// CODESYS_Control_for_Raspberry_Pi/Application/visualization/ups_s2/ups_s2_m3_state
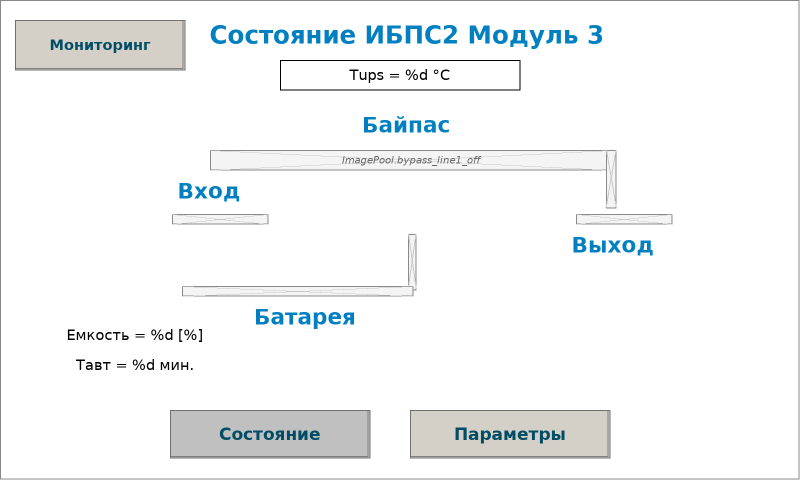
VISUALIZATION ups_s2_m3_state  // 800x480, background image ImagePool.mpx_state_bg
    Rectangle (204,20 406x30), "Состояние ИБПС2 Модуль 3"
    Button (410,410 200x48), "Параметры"
        OnMouseClick:  Assign=ups_s2_m3_params, Type=Assignment
    Button (170,410 200x48), "Состояние", pressed state: PLC_PRG.var_true
    Rectangle (350,110 112x30), "Байпас"
    Rectangle (246,302 118x30), "Батарея"
    Rectangle (166,176 86x30), "Вход"
    Rectangle (560,230 106x30), "Выход"
    Rectangle (280,60 240x30), "Tups = %d °С", text variable: PLC_PRG.mpx_s2_3_temp
    Rectangle (30,320 210x30), "Емкость = %d [%]", text variable: PLC_PRG.mpx_s2_3_battery_capacity
    Rectangle (30,350 210x30), "Tавт = %d мин.", text variable: PLC_PRG.mpx_s2_3_battery_time
    Image (210,150 402x20), image: ImagePool.bypass_line1_off
        p84334746: PLC_PRG.mpx_s2_3_bypass_line_state
    Image (606,150 10x58), image: ImagePool.bypass_arrow_off
        p84334746: PLC_PRG.mpx_s2_3_bypass_arrow_state
    Image (576,214 96x10), image: ImagePool.arrow_off
        p84334746: PLC_PRG.mpx_s2_3_output_state
    Image (172,214 96x10), image: ImagePool.arrow_off
        p84334746: PLC_PRG.mpx_s2_3_input_state
    Image (408,234 8x56), image: ImagePool.battery_arrow_off
        p84334746: PLC_PRG.mpx_s2_3_battery_arrow_state
    Image (182,286 231x10), image: ImagePool.battery_line_off
        p84334746: PLC_PRG.mpx_s2_3_battery_line_state
    Button (15,20 170x50), "Мониторинг"
        OnMouseClick:  Assign=monitoring, Type=Assignment
    hotkey  Id=481037385728, Key=KeyDown=True, KeyName=0, VisuElemId=38
    hotkey  Id=481038434304, Key=KeyName=0, VisuElemId=38
END_VISUALIZATION

// CODESYS_Control_for_Raspberry_Pi/Application/visualization/ups_s1/ups_s1
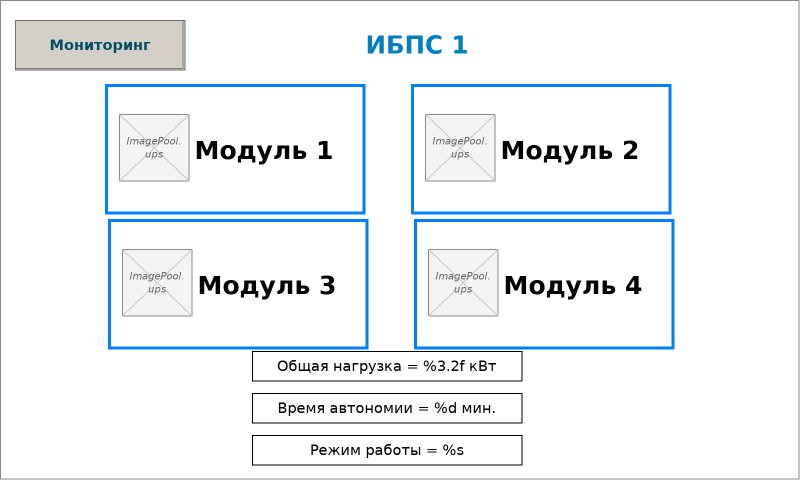
VISUALIZATION ups_s1  // 800x480, background image ImagePool.bg_800
    Group (108,219 260x115)
        OnMouseClick:  Assign=ups_s1_m3_state, Type=Assignment
        RoundedRectangle (0,0 260x130), colour toggle: InterviewState.MPX_S1_3_State
        Image (14,30 70x67), image: ImagePool.ups
        RoundedRectangle (80,38 158x56), "Модуль 3"
            OnMouseClick:  Assign=ups_s2_m1_state, Type=Assignment
    Group (105,84 260x115)
        OnMouseClick:  Assign=ups_s1_m1_state, Type=Assignment
        RoundedRectangle (0,0 260x130), colour toggle: InterviewState.MPX_S1_1_State
        Image (14,30 70x67), image: ImagePool.ups
        RoundedRectangle (80,38 158x56), "Модуль 1"
            OnMouseClick:  Assign=ups_s2_m1_state, Type=Assignment
    Group (414,219 260x115)
        OnMouseClick:  Assign=ups_s1_m4_state, Type=Assignment
        RoundedRectangle (0,0 260x130), colour toggle: InterviewState.MPX_S1_4_State
        Image (14,30 70x67), image: ImagePool.ups
        RoundedRectangle (80,38 158x56), "Модуль 4"
            OnMouseClick:  Assign=ups_s2_m1_state, Type=Assignment
    Group (411,84 260x115)
        OnMouseClick:  Assign=ups_s1_m2_state, Type=Assignment
        RoundedRectangle (0,0 260x130), colour toggle: InterviewState.MPX_S1_2_State
        Image (14,30 70x67), image: ImagePool.ups
        RoundedRectangle (80,38 158x56), "Модуль 2"
            OnMouseClick:  Assign=ups_s2_m1_state, Type=Assignment
    Rectangle (214,30 406x30), "ИБПС 1"
    Button (15,20 170x50), "Мониторинг"
        OnMouseClick:  Assign=monitoring, Type=Assignment
    Rectangle (252,351 270x30), "Общая нагрузка = %3.2f кВт", text variable: PLC_PRG.mpx_s1_all_power
    Rectangle (252,393 270x30), "Время автономии = %d мин.", text variable: PLC_PRG.mpx_s1_1_battery_time
    Rectangle (252,435 270x30), "Режим работы = %s", text variable: PLC_PRG.mpx_s1_state_string
    hotkey  Id=481037385728, Key=KeyDown=True, KeyName=0, VisuElemId=38
    hotkey  Id=481038434304, Key=KeyName=0, VisuElemId=38
END_VISUALIZATION

// CODESYS_Control_for_Raspberry_Pi/Application/visualization/ups_s1/ups_s1_m1_params
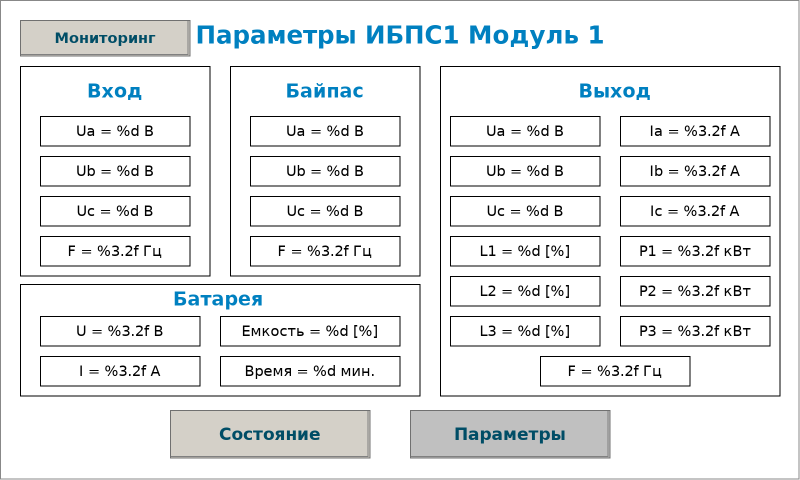
VISUALIZATION ups_s1_m1_params  // 800x480, background image ImagePool.bg_800
    Rectangle (186,20 428x30), "Параметры ИБПC1 Модуль 1"
    Button (170,410 200x48), "Состояние"
        OnMouseClick:  Assign=ups_s1_m1_state, Type=Assignment
    Button (410,410 200x48), "Параметры", pressed state: PLC_PRG.var_true
    Button (20,20 170x36), "Мониторинг"
        OnMouseClick:  Assign=monitoring, Type=Assignment
    Rectangle (20,66 190x210)
    Rectangle (440,66 340x330)
    Rectangle (30,76 170x30), "Вход"
    Rectangle (40,116 150x30), "Ua = %d В", text variable: PLC_PRG.mpx_s1_1_in_v_1
    Rectangle (40,156 150x30), "Ub = %d В", text variable: PLC_PRG.mpx_s1_1_in_v_2
    Rectangle (40,196 150x30), "Uc = %d В", text variable: PLC_PRG.mpx_s1_1_in_v_3
    Rectangle (40,236 150x30), "F = %3.2f Гц", text variable: PLC_PRG.mpx_s1_1_in_freq_real
    Rectangle (230,66 190x210)
    Rectangle (240,76 170x30), "Байпас"
    Rectangle (250,116 150x30), "Ua = %d В", text variable: PLC_PRG.mpx_s1_1_bypass_v_1
    Rectangle (250,156 150x30), "Ub = %d В", text variable: PLC_PRG.mpx_s1_1_bypass_v_2
    Rectangle (250,196 150x30), "Uc = %d В", text variable: PLC_PRG.mpx_s1_1_bypass_v_3
    Rectangle (250,236 150x30), "F = %3.2f Гц", text variable: PLC_PRG.mpx_s1_1_bypass_freq_real
    Rectangle (460,76 310x30), "Выход"
    Rectangle (450,116 150x30), "Ua = %d В", text variable: PLC_PRG.mpx_s1_1_output_v_1
    Rectangle (450,156 150x30), "Ub = %d В", text variable: PLC_PRG.mpx_s1_1_output_v_2
    Rectangle (450,196 150x30), "Uc = %d В", text variable: PLC_PRG.mpx_s1_1_output_v_3
    Rectangle (620,116 150x30), "Ia = %3.2f A", text variable: PLC_PRG.mpx_s1_1_output_i_1_real
    Rectangle (620,156 150x30), "Ib = %3.2f A", text variable: PLC_PRG.mpx_s1_1_output_i_2_real
    Rectangle (620,196 150x30), "Ic = %3.2f A", text variable: PLC_PRG.mpx_s1_1_output_i_3_real
    Rectangle (450,236 150x30), "L1 = %d [%]", text variable: PLC_PRG.mpx_s1_1_load_ph_1
    Rectangle (450,276 150x30), "L2 = %d [%]", text variable: PLC_PRG.mpx_s1_1_load_ph_2
    Rectangle (450,316 150x30), "L3 = %d [%]", text variable: PLC_PRG.mpx_s1_1_load_ph_3
    Rectangle (620,236 150x30), "P1 = %3.2f кВт", text variable: PLC_PRG.mpx_s1_1_output_active_power_1_real
    Rectangle (620,276 150x30), "P2 = %3.2f кВт", text variable: PLC_PRG.mpx_s1_1_output_active_power_2_real
    Rectangle (620,316 150x30), "P3 = %3.2f кВт", text variable: PLC_PRG.mpx_s1_1_output_active_power_3_real
    Rectangle (540,356 150x30), "F = %3.2f Гц", text variable: PLC_PRG.mpx_s1_1_output_freq_real
    Rectangle (20,284 400x112)
    Rectangle (30,290 376x18), "Батарея"
    Rectangle (40,316 160x30), "U = %3.2f В", text variable: PLC_PRG.mpx_s1_1_battery_voltage_real
    Rectangle (40,356 160x30), "I = %3.2f A", text variable: PLC_PRG.mpx_s1_1_battery_current_real
    Rectangle (220,316 180x30), "Емкость = %d [%]", text variable: PLC_PRG.mpx_s1_1_battery_capacity
    Rectangle (220,356 180x30), "Время = %d мин.", text variable: PLC_PRG.mpx_s1_1_battery_time
    hotkey  Id=481037385728, Key=KeyDown=True, KeyName=0, VisuElemId=7
    hotkey  Id=481038434304, Key=KeyName=0, VisuElemId=7
END_VISUALIZATION

// CODESYS_Control_for_Raspberry_Pi/Application/visualization/ups_s1/ups_s1_m1_state
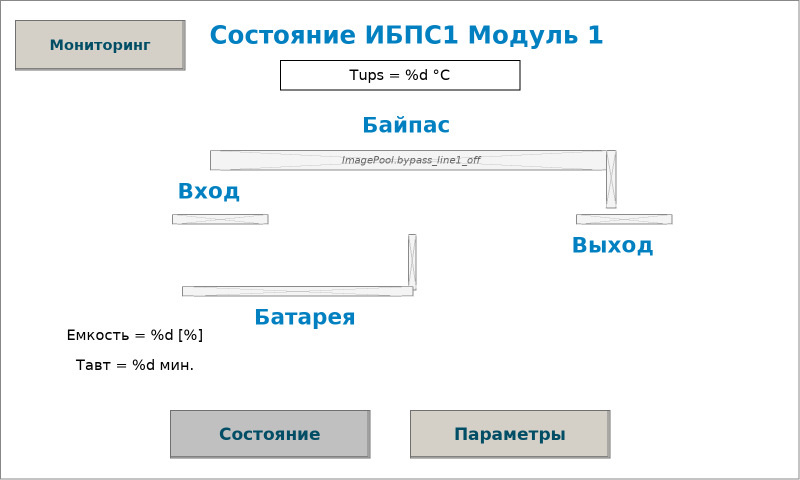
VISUALIZATION ups_s1_m1_state  // 800x480, background image ImagePool.mpx_state_bg
    Rectangle (204,20 406x30), "Состояние ИБПС1 Модуль 1"
    Button (410,410 200x48), "Параметры"
        OnMouseClick:  Assign=ups_s1_m1_params, Type=Assignment
    Button (170,410 200x48), "Состояние", pressed state: PLC_PRG.var_true
    Rectangle (350,110 112x30), "Байпас"
    Rectangle (246,302 118x30), "Батарея"
    Rectangle (166,176 86x30), "Вход"
    Rectangle (560,230 106x30), "Выход"
    Rectangle (280,60 240x30), "Tups = %d °С", text variable: PLC_PRG.mpx_s1_1_temp
    Rectangle (30,320 210x30), "Емкость = %d [%]", text variable: PLC_PRG.mpx_s1_1_battery_capacity
    Rectangle (30,350 210x30), "Tавт = %d мин.", text variable: PLC_PRG.mpx_s1_1_battery_time
    Image (210,150 402x20), image: ImagePool.bypass_line1_off
        p84334746: PLC_PRG.mpx_s1_1_bypass_line_state
    Image (606,150 10x58), image: ImagePool.bypass_arrow_off
        p84334746: PLC_PRG.mpx_s1_1_bypass_arrow_state
    Image (576,214 96x10), image: ImagePool.arrow_off
        p84334746: PLC_PRG.mpx_s1_1_output_state
    Image (172,214 96x10), image: ImagePool.arrow_off
        p84334746: PLC_PRG.mpx_s1_1_input_state
    Image (408,234 8x56), image: ImagePool.battery_arrow_off
        p84334746: PLC_PRG.mpx_s1_1_battery_arrow_state
    Image (182,286 231x10), image: ImagePool.battery_line_off
        p84334746: PLC_PRG.mpx_s1_1_battery_line_state
    Button (15,20 170x50), "Мониторинг"
        OnMouseClick:  Assign=monitoring, Type=Assignment
    hotkey  Id=481037385728, Key=KeyDown=True, KeyName=0, VisuElemId=38
    hotkey  Id=481038434304, Key=KeyName=0, VisuElemId=38
END_VISUALIZATION

// CODESYS_Control_for_Raspberry_Pi/Application/visualization/ups_s1/ups_s1_m2_params
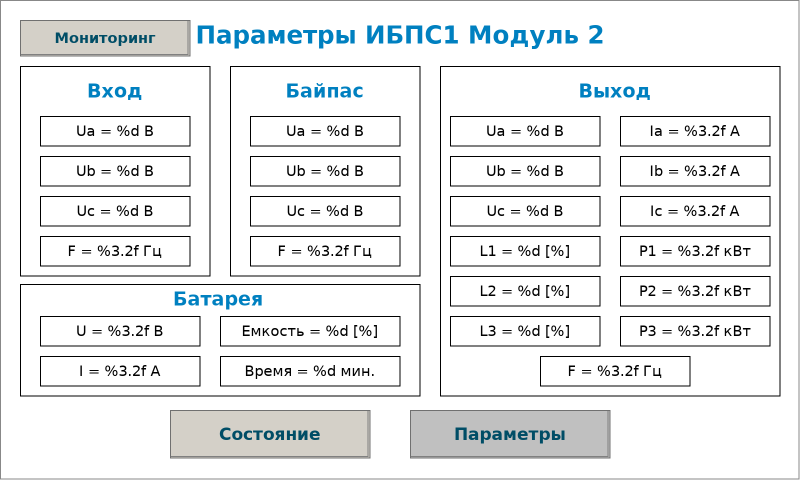
VISUALIZATION ups_s1_m2_params  // 800x480, background image ImagePool.bg_800
    Rectangle (186,20 428x30), "Параметры ИБПC1 Модуль 2"
    Button (170,410 200x48), "Состояние"
        OnMouseClick:  Assign=ups_s1_m2_state, Type=Assignment
    Button (410,410 200x48), "Параметры", pressed state: PLC_PRG.var_true
    Button (20,20 170x36), "Мониторинг"
        OnMouseClick:  Assign=monitoring, Type=Assignment
    Rectangle (20,66 190x210)
    Rectangle (440,66 340x330)
    Rectangle (30,76 170x30), "Вход"
    Rectangle (40,116 150x30), "Ua = %d В", text variable: PLC_PRG.mpx_s1_2_in_v_1
    Rectangle (40,156 150x30), "Ub = %d В", text variable: PLC_PRG.mpx_s1_2_in_v_2
    Rectangle (40,196 150x30), "Uc = %d В", text variable: PLC_PRG.mpx_s1_2_in_v_3
    Rectangle (40,236 150x30), "F = %3.2f Гц", text variable: PLC_PRG.mpx_s1_2_in_freq_real
    Rectangle (230,66 190x210)
    Rectangle (240,76 170x30), "Байпас"
    Rectangle (250,116 150x30), "Ua = %d В", text variable: PLC_PRG.mpx_s1_2_bypass_v_1
    Rectangle (250,156 150x30), "Ub = %d В", text variable: PLC_PRG.mpx_s1_2_bypass_v_2
    Rectangle (250,196 150x30), "Uc = %d В", text variable: PLC_PRG.mpx_s1_2_bypass_v_3
    Rectangle (250,236 150x30), "F = %3.2f Гц", text variable: PLC_PRG.mpx_s1_2_bypass_freq_real
    Rectangle (460,76 310x30), "Выход"
    Rectangle (450,116 150x30), "Ua = %d В", text variable: PLC_PRG.mpx_s1_2_output_v_1
    Rectangle (450,156 150x30), "Ub = %d В", text variable: PLC_PRG.mpx_s1_2_output_v_2
    Rectangle (450,196 150x30), "Uc = %d В", text variable: PLC_PRG.mpx_s1_2_output_v_3
    Rectangle (620,116 150x30), "Ia = %3.2f A", text variable: PLC_PRG.mpx_s1_2_output_i_1_real
    Rectangle (620,156 150x30), "Ib = %3.2f A", text variable: PLC_PRG.mpx_s1_2_output_i_2_real
    Rectangle (620,196 150x30), "Ic = %3.2f A", text variable: PLC_PRG.mpx_s1_2_output_i_3_real
    Rectangle (450,236 150x30), "L1 = %d [%]", text variable: PLC_PRG.mpx_s1_2_load_ph_1
    Rectangle (450,276 150x30), "L2 = %d [%]", text variable: PLC_PRG.mpx_s1_2_load_ph_2
    Rectangle (450,316 150x30), "L3 = %d [%]", text variable: PLC_PRG.mpx_s1_2_load_ph_3
    Rectangle (620,236 150x30), "P1 = %3.2f кВт", text variable: PLC_PRG.mpx_s1_2_output_active_power_1_real
    Rectangle (620,276 150x30), "P2 = %3.2f кВт", text variable: PLC_PRG.mpx_s1_2_output_active_power_2_real
    Rectangle (620,316 150x30), "P3 = %3.2f кВт", text variable: PLC_PRG.mpx_s1_2_output_active_power_3_real
    Rectangle (540,356 150x30), "F = %3.2f Гц", text variable: PLC_PRG.mpx_s1_2_output_freq_real
    Rectangle (20,284 400x112)
    Rectangle (30,290 376x18), "Батарея"
    Rectangle (40,316 160x30), "U = %3.2f В", text variable: PLC_PRG.mpx_s1_2_battery_voltage_real
    Rectangle (40,356 160x30), "I = %3.2f A", text variable: PLC_PRG.mpx_s1_2_battery_current_real
    Rectangle (220,316 180x30), "Емкость = %d [%]", text variable: PLC_PRG.mpx_s1_2_battery_capacity
    Rectangle (220,356 180x30), "Время = %d мин.", text variable: PLC_PRG.mpx_s1_2_battery_time
    hotkey  Id=481037385728, Key=KeyDown=True, KeyName=0, VisuElemId=7
    hotkey  Id=481038434304, Key=KeyName=0, VisuElemId=7
END_VISUALIZATION

// CODESYS_Control_for_Raspberry_Pi/Application/visualization/ups_s1/ups_s1_m2_state
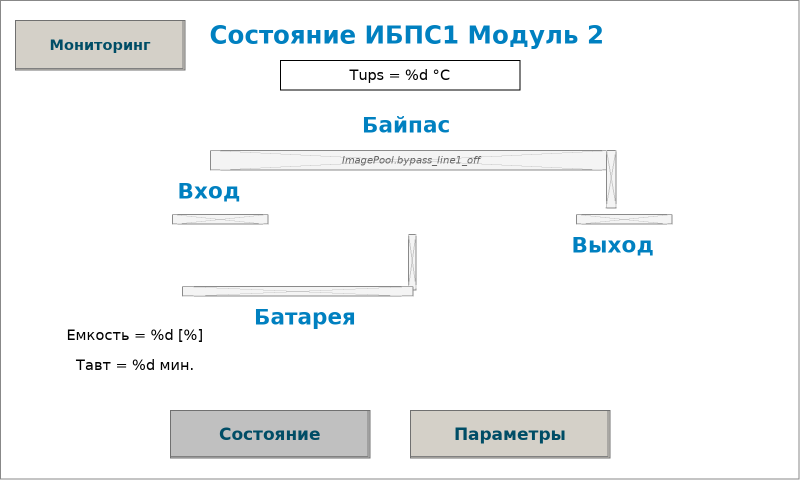
VISUALIZATION ups_s1_m2_state  // 800x480, background image ImagePool.mpx_state_bg
    Rectangle (204,20 406x30), "Состояние ИБПС1 Модуль 2"
    Button (410,410 200x48), "Параметры"
        OnMouseClick:  Assign=ups_s1_m2_params, Type=Assignment
    Button (170,410 200x48), "Состояние", pressed state: PLC_PRG.var_true
    Rectangle (350,110 112x30), "Байпас"
    Rectangle (246,302 118x30), "Батарея"
    Rectangle (166,176 86x30), "Вход"
    Rectangle (560,230 106x30), "Выход"
    Rectangle (280,60 240x30), "Tups = %d °С", text variable: PLC_PRG.mpx_s1_2_temp
    Rectangle (30,320 210x30), "Емкость = %d [%]", text variable: PLC_PRG.mpx_s1_2_battery_capacity
    Rectangle (30,350 210x30), "Tавт = %d мин.", text variable: PLC_PRG.mpx_s1_2_battery_time
    Image (210,150 402x20), image: ImagePool.bypass_line1_off
        p84334746: PLC_PRG.mpx_s1_2_bypass_line_state
    Image (606,150 10x58), image: ImagePool.bypass_arrow_off
        p84334746: PLC_PRG.mpx_s1_2_bypass_arrow_state
    Image (576,214 96x10), image: ImagePool.arrow_off
        p84334746: PLC_PRG.mpx_s1_2_output_state
    Image (172,214 96x10), image: ImagePool.arrow_off
        p84334746: PLC_PRG.mpx_s1_2_input_state
    Image (408,234 8x56), image: ImagePool.battery_arrow_off
        p84334746: PLC_PRG.mpx_s1_2_battery_arrow_state
    Image (182,286 231x10), image: ImagePool.battery_line_off
        p84334746: PLC_PRG.mpx_s1_2_battery_line_state
    Button (15,20 170x50), "Мониторинг"
        OnMouseClick:  Assign=monitoring, Type=Assignment
    hotkey  Id=481037385728, Key=KeyDown=True, KeyName=0, VisuElemId=38
    hotkey  Id=481038434304, Key=KeyName=0, VisuElemId=38
END_VISUALIZATION

// CODESYS_Control_for_Raspberry_Pi/Application/visualization/ups_s1/ups_s1_m3_params
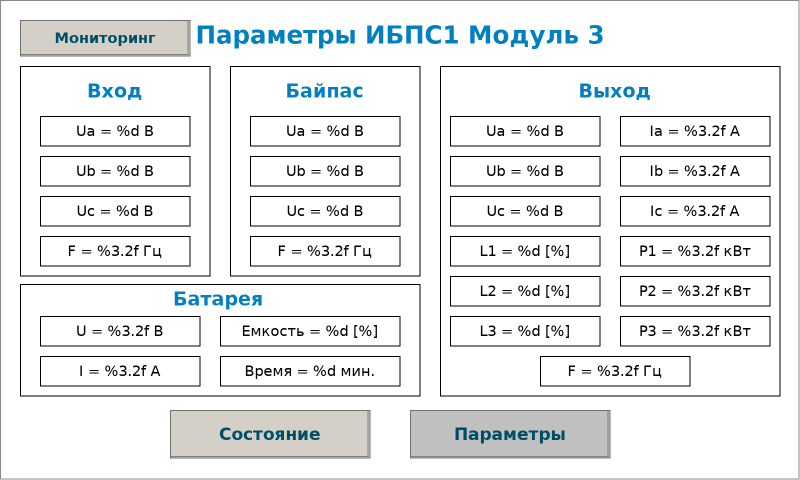
VISUALIZATION ups_s1_m3_params  // 800x480, background image ImagePool.bg_800
    Rectangle (186,20 428x30), "Параметры ИБПC1 Модуль 3"
    Button (170,410 200x48), "Состояние"
        OnMouseClick:  Assign=ups_s1_m3_state, Type=Assignment
    Button (410,410 200x48), "Параметры", pressed state: PLC_PRG.var_true
    Button (20,20 170x36), "Мониторинг"
        OnMouseClick:  Assign=monitoring, Type=Assignment
    Rectangle (20,66 190x210)
    Rectangle (440,66 340x330)
    Rectangle (30,76 170x30), "Вход"
    Rectangle (40,116 150x30), "Ua = %d В", text variable: PLC_PRG.mpx_s1_3_in_v_1
    Rectangle (40,156 150x30), "Ub = %d В", text variable: PLC_PRG.mpx_s1_3_in_v_2
    Rectangle (40,196 150x30), "Uc = %d В", text variable: PLC_PRG.mpx_s1_3_in_v_3
    Rectangle (40,236 150x30), "F = %3.2f Гц", text variable: PLC_PRG.mpx_s1_3_in_freq_real
    Rectangle (230,66 190x210)
    Rectangle (240,76 170x30), "Байпас"
    Rectangle (250,116 150x30), "Ua = %d В", text variable: PLC_PRG.mpx_s1_3_bypass_v_1
    Rectangle (250,156 150x30), "Ub = %d В", text variable: PLC_PRG.mpx_s1_3_bypass_v_2
    Rectangle (250,196 150x30), "Uc = %d В", text variable: PLC_PRG.mpx_s1_3_bypass_v_3
    Rectangle (250,236 150x30), "F = %3.2f Гц", text variable: PLC_PRG.mpx_s1_3_bypass_freq_real
    Rectangle (460,76 310x30), "Выход"
    Rectangle (450,116 150x30), "Ua = %d В", text variable: PLC_PRG.mpx_s1_3_output_v_1
    Rectangle (450,156 150x30), "Ub = %d В", text variable: PLC_PRG.mpx_s1_3_output_v_2
    Rectangle (450,196 150x30), "Uc = %d В", text variable: PLC_PRG.mpx_s1_3_output_v_3
    Rectangle (620,116 150x30), "Ia = %3.2f A", text variable: PLC_PRG.mpx_s1_3_output_i_1_real
    Rectangle (620,156 150x30), "Ib = %3.2f A", text variable: PLC_PRG.mpx_s1_3_output_i_2_real
    Rectangle (620,196 150x30), "Ic = %3.2f A", text variable: PLC_PRG.mpx_s1_3_output_i_3_real
    Rectangle (450,236 150x30), "L1 = %d [%]", text variable: PLC_PRG.mpx_s1_3_load_ph_1
    Rectangle (450,276 150x30), "L2 = %d [%]", text variable: PLC_PRG.mpx_s1_3_load_ph_2
    Rectangle (450,316 150x30), "L3 = %d [%]", text variable: PLC_PRG.mpx_s1_3_load_ph_3
    Rectangle (620,236 150x30), "P1 = %3.2f кВт", text variable: PLC_PRG.mpx_s1_3_output_active_power_1_real
    Rectangle (620,276 150x30), "P2 = %3.2f кВт", text variable: PLC_PRG.mpx_s1_3_output_active_power_2_real
    Rectangle (620,316 150x30), "P3 = %3.2f кВт", text variable: PLC_PRG.mpx_s1_3_output_active_power_3_real
    Rectangle (540,356 150x30), "F = %3.2f Гц", text variable: PLC_PRG.mpx_s1_3_output_freq_real
    Rectangle (20,284 400x112)
    Rectangle (30,290 376x18), "Батарея"
    Rectangle (40,316 160x30), "U = %3.2f В", text variable: PLC_PRG.mpx_s1_3_battery_voltage_real
    Rectangle (40,356 160x30), "I = %3.2f A", text variable: PLC_PRG.mpx_s1_3_battery_current_real
    Rectangle (220,316 180x30), "Емкость = %d [%]", text variable: PLC_PRG.mpx_s1_3_battery_capacity
    Rectangle (220,356 180x30), "Время = %d мин.", text variable: PLC_PRG.mpx_s1_3_battery_time
    hotkey  Id=481037385728, Key=KeyDown=True, KeyName=0, VisuElemId=7
    hotkey  Id=481038434304, Key=KeyName=0, VisuElemId=7
END_VISUALIZATION

// CODESYS_Control_for_Raspberry_Pi/Application/visualization/ups_s1/ups_s1_m3_state
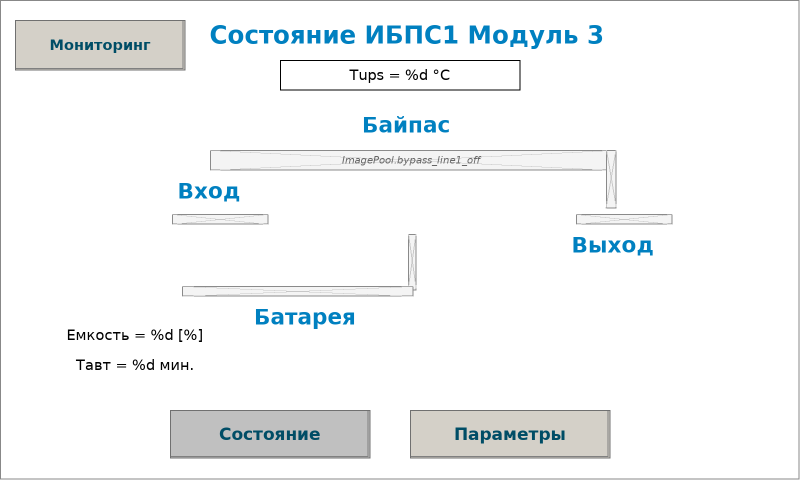
VISUALIZATION ups_s1_m3_state  // 800x480, background image ImagePool.mpx_state_bg
    Rectangle (204,20 406x30), "Состояние ИБПС1 Модуль 3"
    Button (410,410 200x48), "Параметры"
        OnMouseClick:  Assign=ups_s1_m3_params, Type=Assignment
    Button (170,410 200x48), "Состояние", pressed state: PLC_PRG.var_true
    Rectangle (350,110 112x30), "Байпас"
    Rectangle (246,302 118x30), "Батарея"
    Rectangle (166,176 86x30), "Вход"
    Rectangle (560,230 106x30), "Выход"
    Rectangle (280,60 240x30), "Tups = %d °С", text variable: PLC_PRG.mpx_s1_3_temp
    Rectangle (30,320 210x30), "Емкость = %d [%]", text variable: PLC_PRG.mpx_s1_3_battery_capacity
    Rectangle (30,350 210x30), "Tавт = %d мин.", text variable: PLC_PRG.mpx_s1_3_battery_time
    Image (210,150 402x20), image: ImagePool.bypass_line1_off
        p84334746: PLC_PRG.mpx_s1_3_bypass_line_state
    Image (606,150 10x58), image: ImagePool.bypass_arrow_off
        p84334746: PLC_PRG.mpx_s1_3_bypass_arrow_state
    Image (576,214 96x10), image: ImagePool.arrow_off
        p84334746: PLC_PRG.mpx_s1_3_output_state
    Image (172,214 96x10), image: ImagePool.arrow_off
        p84334746: PLC_PRG.mpx_s1_3_input_state
    Image (408,234 8x56), image: ImagePool.battery_arrow_off
        p84334746: PLC_PRG.mpx_s1_3_battery_arrow_state
    Image (182,286 231x10), image: ImagePool.battery_line_off
        p84334746: PLC_PRG.mpx_s1_3_battery_line_state
    Button (15,20 170x50), "Мониторинг"
        OnMouseClick:  Assign=monitoring, Type=Assignment
    hotkey  Id=481037385728, Key=KeyDown=True, KeyName=0, VisuElemId=38
    hotkey  Id=481038434304, Key=KeyName=0, VisuElemId=38
END_VISUALIZATION

// CODESYS_Control_for_Raspberry_Pi/Application/visualization/ups_s1/ups_s1_m4_params
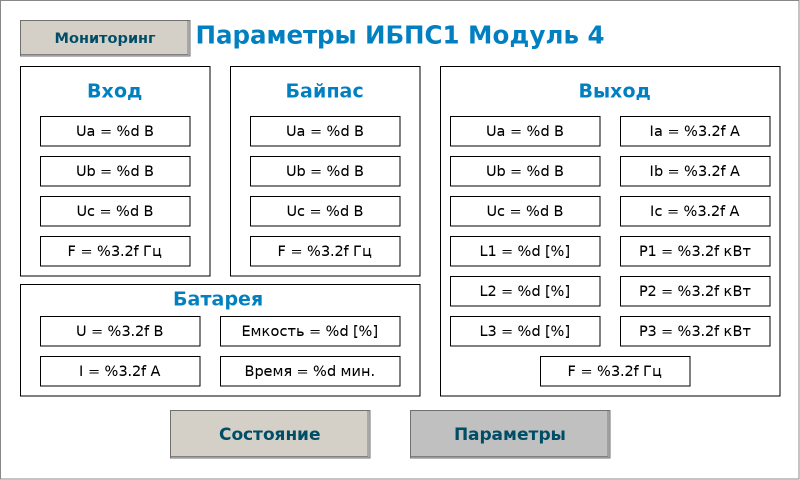
VISUALIZATION ups_s1_m4_params  // 800x480, background image ImagePool.bg_800
    Rectangle (186,20 428x30), "Параметры ИБПC1 Модуль 4"
    Button (170,410 200x48), "Состояние"
        OnMouseClick:  Assign=ups_s1_m4_state, Type=Assignment
    Button (410,410 200x48), "Параметры", pressed state: PLC_PRG.var_true
    Button (20,20 170x36), "Мониторинг"
        OnMouseClick:  Assign=monitoring, Type=Assignment
    Rectangle (20,66 190x210)
    Rectangle (440,66 340x330)
    Rectangle (30,76 170x30), "Вход"
    Rectangle (40,116 150x30), "Ua = %d В", text variable: PLC_PRG.mpx_s1_4_in_v_1
    Rectangle (40,156 150x30), "Ub = %d В", text variable: PLC_PRG.mpx_s1_4_in_v_2
    Rectangle (40,196 150x30), "Uc = %d В", text variable: PLC_PRG.mpx_s1_4_in_v_3
    Rectangle (40,236 150x30), "F = %3.2f Гц", text variable: PLC_PRG.mpx_s1_4_in_freq_real
    Rectangle (230,66 190x210)
    Rectangle (240,76 170x30), "Байпас"
    Rectangle (250,116 150x30), "Ua = %d В", text variable: PLC_PRG.mpx_s1_4_bypass_v_1
    Rectangle (250,156 150x30), "Ub = %d В", text variable: PLC_PRG.mpx_s1_4_bypass_v_2
    Rectangle (250,196 150x30), "Uc = %d В", text variable: PLC_PRG.mpx_s1_4_bypass_v_3
    Rectangle (250,236 150x30), "F = %3.2f Гц", text variable: PLC_PRG.mpx_s1_4_bypass_freq_real
    Rectangle (460,76 310x30), "Выход"
    Rectangle (450,116 150x30), "Ua = %d В", text variable: PLC_PRG.mpx_s1_4_output_v_1
    Rectangle (450,156 150x30), "Ub = %d В", text variable: PLC_PRG.mpx_s1_4_output_v_2
    Rectangle (450,196 150x30), "Uc = %d В", text variable: PLC_PRG.mpx_s1_4_output_v_3
    Rectangle (620,116 150x30), "Ia = %3.2f A", text variable: PLC_PRG.mpx_s1_4_output_i_1_real
    Rectangle (620,156 150x30), "Ib = %3.2f A", text variable: PLC_PRG.mpx_s1_4_output_i_2_real
    Rectangle (620,196 150x30), "Ic = %3.2f A", text variable: PLC_PRG.mpx_s1_4_output_i_3_real
    Rectangle (450,236 150x30), "L1 = %d [%]", text variable: PLC_PRG.mpx_s1_4_load_ph_1
    Rectangle (450,276 150x30), "L2 = %d [%]", text variable: PLC_PRG.mpx_s1_4_load_ph_2
    Rectangle (450,316 150x30), "L3 = %d [%]", text variable: PLC_PRG.mpx_s1_4_load_ph_3
    Rectangle (620,236 150x30), "P1 = %3.2f кВт", text variable: PLC_PRG.mpx_s1_4_output_active_power_1_real
    Rectangle (620,276 150x30), "P2 = %3.2f кВт", text variable: PLC_PRG.mpx_s1_4_output_active_power_2_real
    Rectangle (620,316 150x30), "P3 = %3.2f кВт", text variable: PLC_PRG.mpx_s1_4_output_active_power_3_real
    Rectangle (540,356 150x30), "F = %3.2f Гц", text variable: PLC_PRG.mpx_s1_4_output_freq_real
    Rectangle (20,284 400x112)
    Rectangle (30,290 376x18), "Батарея"
    Rectangle (40,316 160x30), "U = %3.2f В", text variable: PLC_PRG.mpx_s1_4_battery_voltage_real
    Rectangle (40,356 160x30), "I = %3.2f A", text variable: PLC_PRG.mpx_s1_4_battery_current_real
    Rectangle (220,316 180x30), "Емкость = %d [%]", text variable: PLC_PRG.mpx_s1_4_battery_capacity
    Rectangle (220,356 180x30), "Время = %d мин.", text variable: PLC_PRG.mpx_s1_4_battery_time
    hotkey  Id=481037385728, Key=KeyDown=True, KeyName=0, VisuElemId=7
    hotkey  Id=481038434304, Key=KeyName=0, VisuElemId=7
END_VISUALIZATION

// CODESYS_Control_for_Raspberry_Pi/Application/visualization/ups_s1/ups_s1_m4_state
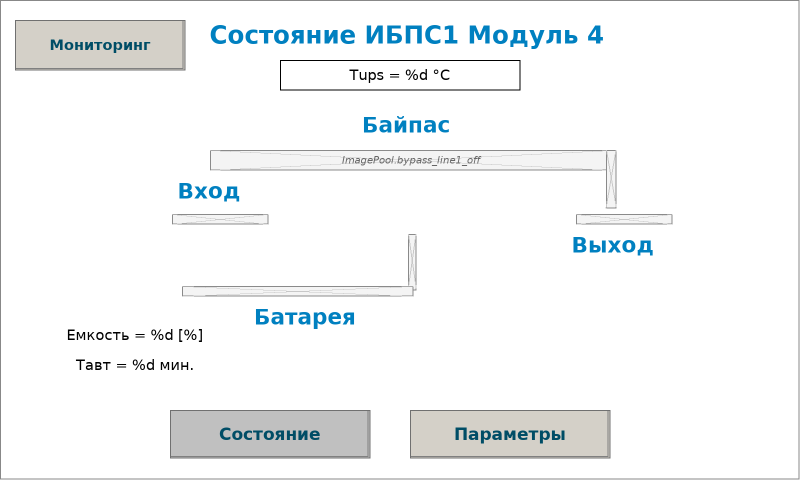
VISUALIZATION ups_s1_m4_state  // 800x480, background image ImagePool.mpx_state_bg
    Rectangle (204,20 406x30), "Состояние ИБПС1 Модуль 4"
    Button (410,410 200x48), "Параметры"
        OnMouseClick:  Assign=ups_s1_m4_params, Type=Assignment
    Button (170,410 200x48), "Состояние", pressed state: PLC_PRG.var_true
    Rectangle (350,110 112x30), "Байпас"
    Rectangle (246,302 118x30), "Батарея"
    Rectangle (166,176 86x30), "Вход"
    Rectangle (560,230 106x30), "Выход"
    Rectangle (280,60 240x30), "Tups = %d °С", text variable: PLC_PRG.mpx_s1_4_temp
    Rectangle (30,320 210x30), "Емкость = %d [%]", text variable: PLC_PRG.mpx_s1_4_battery_capacity
    Rectangle (30,350 210x30), "Tавт = %d мин.", text variable: PLC_PRG.mpx_s1_4_battery_time
    Image (210,150 402x20), image: ImagePool.bypass_line1_off
        p84334746: PLC_PRG.mpx_s1_4_bypass_line_state
    Image (606,150 10x58), image: ImagePool.bypass_arrow_off
        p84334746: PLC_PRG.mpx_s1_4_bypass_arrow_state
    Image (576,214 96x10), image: ImagePool.arrow_off
        p84334746: PLC_PRG.mpx_s1_4_output_state
    Image (172,214 96x10), image: ImagePool.arrow_off
        p84334746: PLC_PRG.mpx_s1_4_input_state
    Image (408,234 8x56), image: ImagePool.battery_arrow_off
        p84334746: PLC_PRG.mpx_s1_4_battery_arrow_state
    Image (182,286 231x10), image: ImagePool.battery_line_off
        p84334746: PLC_PRG.mpx_s1_4_battery_line_state
    Button (15,20 170x50), "Мониторинг"
        OnMouseClick:  Assign=monitoring, Type=Assignment
    hotkey  Id=481037385728, Key=KeyDown=True, KeyName=0, VisuElemId=38
    hotkey  Id=481038434304, Key=KeyName=0, VisuElemId=38
END_VISUALIZATION

// CODESYS_Control_for_Raspberry_Pi/Application/visualization/ups_a1/ups_a1
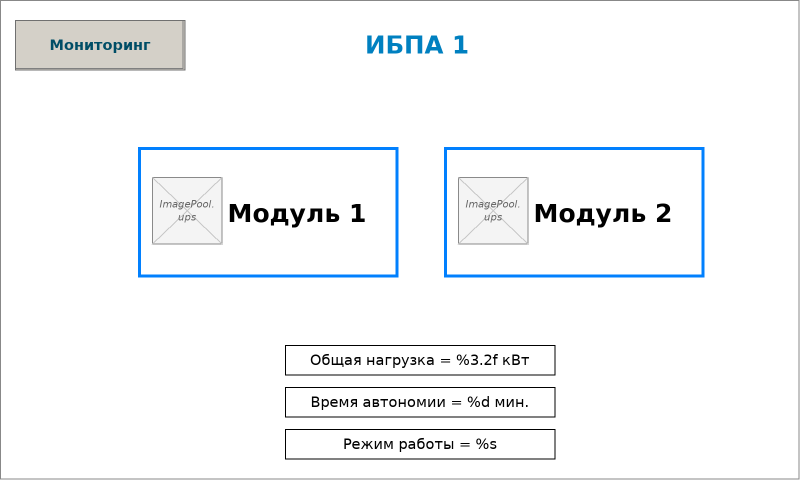
VISUALIZATION ups_a1  // 800x480, background image ImagePool.bg_800
    Rectangle (214,30 406x30), "ИБПА 1"
    Button (15,20 170x50), "Мониторинг"
        OnMouseClick:  Assign=monitoring, Type=Assignment
    Group (138,147 260x115)
        OnMouseClick:  Assign=ups_a1_m1_state, Type=Assignment
        RoundedRectangle (0,0 260x130), colour toggle: InterviewState.MPX_S1_1_State
        Image (14,30 70x67), image: ImagePool.ups
        RoundedRectangle (80,38 158x56), "Модуль 1"
            OnMouseClick:  Assign=ups_s2_m1_state, Type=Assignment
    Group (444,147 260x115)
        OnMouseClick:  Assign=ups_a1_m2_state, Type=Assignment
        RoundedRectangle (0,0 260x130), colour toggle: InterviewState.MPX_S1_2_State
        Image (14,30 70x67), image: ImagePool.ups
        RoundedRectangle (80,38 158x56), "Модуль 2"
            OnMouseClick:  Assign=ups_s2_m1_state, Type=Assignment
    Rectangle (285,345 270x30), "Общая нагрузка = %3.2f кВт", text variable: PLC_PRG.mpx_a1_all_power
    Rectangle (285,387 270x30), "Время автономии = %d мин.", text variable: PLC_PRG.mpx_a1_1_battery_time
    Rectangle (285,429 270x30), "Режим работы = %s", text variable: PLC_PRG.mpx_a1_state_string
    hotkey  Id=481037385728, Key=KeyDown=True, KeyName=0, VisuElemId=38
    hotkey  Id=481038434304, Key=KeyName=0, VisuElemId=38
END_VISUALIZATION

// CODESYS_Control_for_Raspberry_Pi/Application/visualization/ups_a1/ups_a1_m1_params
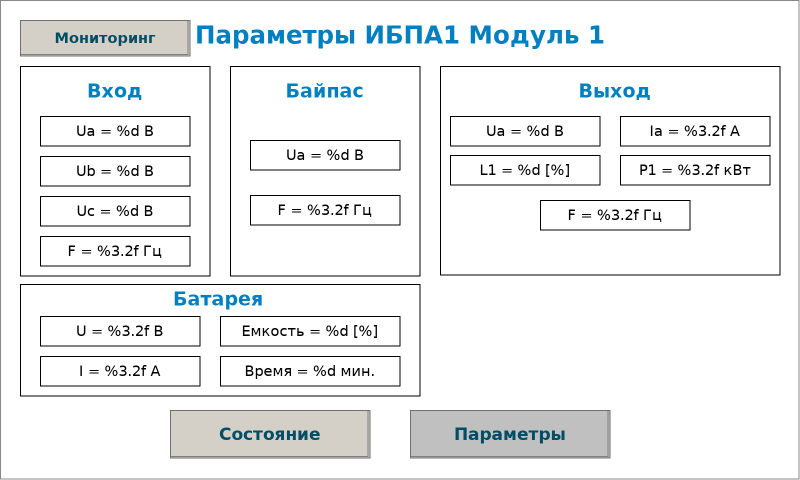
VISUALIZATION ups_a1_m1_params  // 800x480, background image ImagePool.bg_800
    Rectangle (186,20 428x30), "Параметры ИБПА1 Модуль 1"
    Button (170,410 200x48), "Состояние"
        OnMouseClick:  Assign=ups_a1_m1_state, Type=Assignment
    Button (410,410 200x48), "Параметры", pressed state: PLC_PRG.var_true
    Button (20,20 170x36), "Мониторинг"
        OnMouseClick:  Assign=monitoring, Type=Assignment
    Rectangle (20,66 190x210)
    Rectangle (440,66 340x209)
    Rectangle (30,76 170x30), "Вход"
    Rectangle (40,116 150x30), "Ua = %d В", text variable: PLC_PRG.mpx_a1_1_in_v_1
    Rectangle (40,156 150x30), "Ub = %d В", text variable: PLC_PRG.mpx_a1_1_in_v_2
    Rectangle (40,196 150x30), "Uc = %d В", text variable: PLC_PRG.mpx_a1_1_in_v_3
    Rectangle (40,236 150x30), "F = %3.2f Гц", text variable: PLC_PRG.mpx_a1_1_in_freq_real
    Rectangle (230,66 190x210)
    Rectangle (240,76 170x30), "Байпас"
    Rectangle (250,140 150x30), "Ua = %d В", text variable: PLC_PRG.mpx_a1_1_bypass_v_1
    Rectangle (250,195 150x30), "F = %3.2f Гц", text variable: PLC_PRG.mpx_a1_1_bypass_freq_real
    Rectangle (460,76 310x30), "Выход"
    Rectangle (450,116 150x30), "Ua = %d В", text variable: PLC_PRG.mpx_a1_1_output_v_1
    Rectangle (620,116 150x30), "Ia = %3.2f A", text variable: PLC_PRG.mpx_a1_1_output_i_1_real
    Rectangle (450,155 150x30), "L1 = %d [%]", text variable: PLC_PRG.mpx_a1_1_load_ph_1
    Rectangle (620,155 150x30), "P1 = %3.2f кВт", text variable: PLC_PRG.mpx_a1_1_output_active_power_1_real
    Rectangle (540,200 150x30), "F = %3.2f Гц", text variable: PLC_PRG.mpx_a1_1_output_freq_real
    Rectangle (20,284 400x112)
    Rectangle (30,290 376x18), "Батарея"
    Rectangle (40,316 160x30), "U = %3.2f В", text variable: PLC_PRG.mpx_a1_1_battery_voltage_real
    Rectangle (40,356 160x30), "I = %3.2f A", text variable: PLC_PRG.mpx_a1_1_battery_current_real
    Rectangle (220,316 180x30), "Емкость = %d [%]", text variable: PLC_PRG.mpx_a1_1_battery_capacity
    Rectangle (220,356 180x30), "Время = %d мин.", text variable: PLC_PRG.mpx_a1_1_battery_time
    hotkey  Id=481037385728, Key=KeyDown=True, KeyName=0, VisuElemId=7
    hotkey  Id=481038434304, Key=KeyName=0, VisuElemId=7
END_VISUALIZATION

// CODESYS_Control_for_Raspberry_Pi/Application/visualization/ups_a1/ups_a1_m1_state
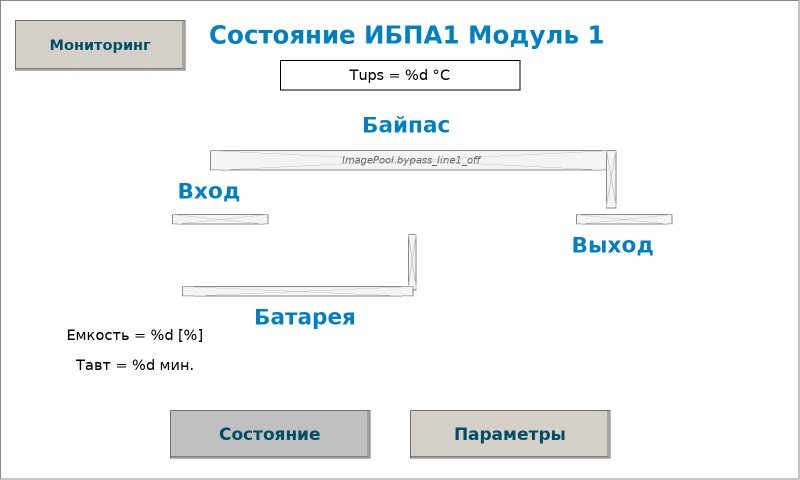
VISUALIZATION ups_a1_m1_state  // 800x480, background image ImagePool.mpx_state_bg
    Rectangle (204,20 406x30), "Состояние ИБПА1 Модуль 1"
    Button (410,410 200x48), "Параметры"
        OnMouseClick:  Assign=ups_a1_m1_params, Type=Assignment
    Button (170,410 200x48), "Состояние", pressed state: PLC_PRG.var_true
    Rectangle (350,110 112x30), "Байпас"
    Rectangle (246,302 118x30), "Батарея"
    Rectangle (166,176 86x30), "Вход"
    Rectangle (560,230 106x30), "Выход"
    Rectangle (280,60 240x30), "Tups = %d °С", text variable: PLC_PRG.mpx_a1_1_temp
    Rectangle (30,320 210x30), "Емкость = %d [%]", text variable: PLC_PRG.mpx_a1_1_battery_capacity
    Rectangle (30,350 210x30), "Tавт = %d мин.", text variable: PLC_PRG.mpx_a1_1_battery_time
    Image (210,150 402x20), image: ImagePool.bypass_line1_off
        p84334746: PLC_PRG.mpx_a1_1_bypass_line_state
    Image (606,150 10x58), image: ImagePool.bypass_arrow_off
        p84334746: PLC_PRG.mpx_a1_1_bypass_arrow_state
    Image (576,214 96x10), image: ImagePool.arrow_off
        p84334746: PLC_PRG.mpx_a1_1_output_state
    Image (172,214 96x10), image: ImagePool.arrow_off
        p84334746: PLC_PRG.mpx_a1_1_input_state
    Image (408,234 8x56), image: ImagePool.battery_arrow_off
        p84334746: PLC_PRG.mpx_a1_1_battery_arrow_state
    Image (182,286 231x10), image: ImagePool.battery_line_off
        p84334746: PLC_PRG.mpx_a1_1_battery_line_state
    Button (15,20 170x50), "Мониторинг"
        OnMouseClick:  Assign=monitoring, Type=Assignment
    hotkey  Id=481037385728, Key=KeyDown=True, KeyName=0, VisuElemId=38
    hotkey  Id=481038434304, Key=KeyName=0, VisuElemId=38
END_VISUALIZATION

// CODESYS_Control_for_Raspberry_Pi/Application/visualization/ups_a1/ups_a1_m2_params
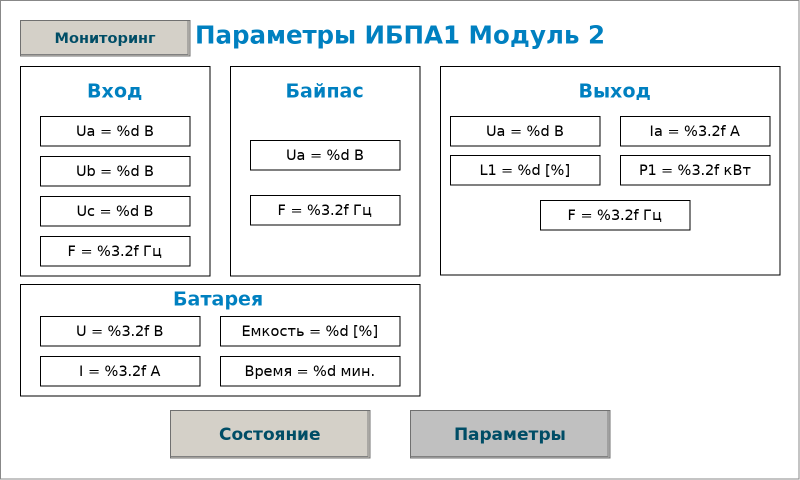
VISUALIZATION ups_a1_m2_params  // 800x480, background image ImagePool.bg_800
    Rectangle (186,20 428x30), "Параметры ИБПА1 Модуль 2"
    Button (170,410 200x48), "Состояние"
        OnMouseClick:  Assign=ups_a1_m2_state, Type=Assignment
    Button (410,410 200x48), "Параметры", pressed state: PLC_PRG.var_true
    Button (20,20 170x36), "Мониторинг"
        OnMouseClick:  Assign=monitoring, Type=Assignment
    Rectangle (20,66 190x210)
    Rectangle (440,66 340x209)
    Rectangle (30,76 170x30), "Вход"
    Rectangle (40,116 150x30), "Ua = %d В", text variable: PLC_PRG.mpx_a1_2_in_v_1
    Rectangle (40,156 150x30), "Ub = %d В", text variable: PLC_PRG.mpx_a1_2_in_v_2
    Rectangle (40,196 150x30), "Uc = %d В", text variable: PLC_PRG.mpx_a1_2_in_v_3
    Rectangle (40,236 150x30), "F = %3.2f Гц", text variable: PLC_PRG.mpx_a1_2_in_freq_real
    Rectangle (230,66 190x210)
    Rectangle (240,76 170x30), "Байпас"
    Rectangle (250,140 150x30), "Ua = %d В", text variable: PLC_PRG.mpx_a1_2_bypass_v_1
    Rectangle (250,195 150x30), "F = %3.2f Гц", text variable: PLC_PRG.mpx_a1_2_bypass_freq_real
    Rectangle (460,76 310x30), "Выход"
    Rectangle (450,116 150x30), "Ua = %d В", text variable: PLC_PRG.mpx_a1_2_output_v_1
    Rectangle (620,116 150x30), "Ia = %3.2f A", text variable: PLC_PRG.mpx_a1_2_output_i_1_real
    Rectangle (450,155 150x30), "L1 = %d [%]", text variable: PLC_PRG.mpx_a1_2_load_ph_1
    Rectangle (620,155 150x30), "P1 = %3.2f кВт", text variable: PLC_PRG.mpx_a1_2_output_active_power_1_real
    Rectangle (540,200 150x30), "F = %3.2f Гц", text variable: PLC_PRG.mpx_a1_2_output_freq_real
    Rectangle (20,284 400x112)
    Rectangle (30,290 376x18), "Батарея"
    Rectangle (40,316 160x30), "U = %3.2f В", text variable: PLC_PRG.mpx_a1_2_battery_voltage_real
    Rectangle (40,356 160x30), "I = %3.2f A", text variable: PLC_PRG.mpx_a1_2_battery_current_real
    Rectangle (220,316 180x30), "Емкость = %d [%]", text variable: PLC_PRG.mpx_a1_2_battery_capacity
    Rectangle (220,356 180x30), "Время = %d мин.", text variable: PLC_PRG.mpx_a1_2_battery_time
    hotkey  Id=481037385728, Key=KeyDown=True, KeyName=0, VisuElemId=7
    hotkey  Id=481038434304, Key=KeyName=0, VisuElemId=7
END_VISUALIZATION

// CODESYS_Control_for_Raspberry_Pi/Application/visualization/ups_a1/ups_a1_m2_state
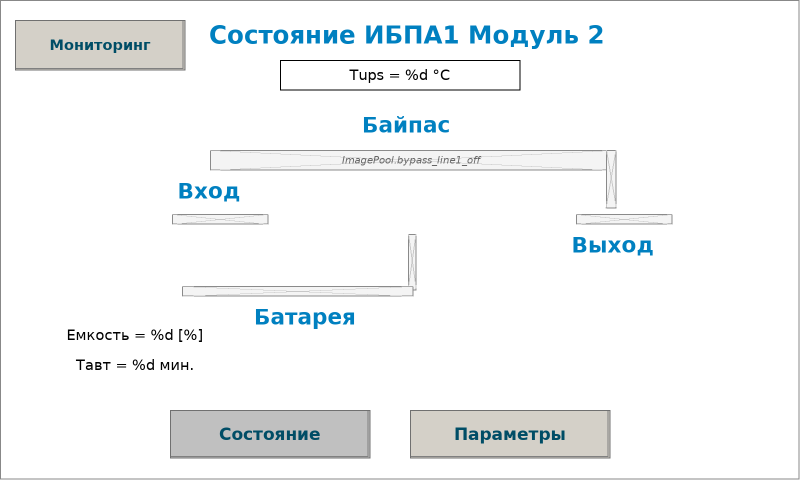
VISUALIZATION ups_a1_m2_state  // 800x480, background image ImagePool.mpx_state_bg
    Rectangle (204,20 406x30), "Состояние ИБПА1 Модуль 2"
    Button (410,410 200x48), "Параметры"
        OnMouseClick:  Assign=ups_a1_m2_params, Type=Assignment
    Button (170,410 200x48), "Состояние", pressed state: PLC_PRG.var_true
    Rectangle (350,110 112x30), "Байпас"
    Rectangle (246,302 118x30), "Батарея"
    Rectangle (166,176 86x30), "Вход"
    Rectangle (560,230 106x30), "Выход"
    Rectangle (280,60 240x30), "Tups = %d °С", text variable: PLC_PRG.mpx_a1_2_temp
    Rectangle (30,320 210x30), "Емкость = %d [%]", text variable: PLC_PRG.mpx_a1_2_battery_capacity
    Rectangle (30,350 210x30), "Tавт = %d мин.", text variable: PLC_PRG.mpx_a1_2_battery_time
    Image (210,150 402x20), image: ImagePool.bypass_line1_off
        p84334746: PLC_PRG.mpx_a1_2_bypass_line_state
    Image (606,150 10x58), image: ImagePool.bypass_arrow_off
        p84334746: PLC_PRG.mpx_a1_2_bypass_arrow_state
    Image (576,214 96x10), image: ImagePool.arrow_off
        p84334746: PLC_PRG.mpx_a1_2_output_state
    Image (172,214 96x10), image: ImagePool.arrow_off
        p84334746: PLC_PRG.mpx_a1_2_input_state
    Image (408,234 8x56), image: ImagePool.battery_arrow_off
        p84334746: PLC_PRG.mpx_a1_2_battery_arrow_state
    Image (182,286 231x10), image: ImagePool.battery_line_off
        p84334746: PLC_PRG.mpx_a1_2_battery_line_state
    Button (15,20 170x50), "Мониторинг"
        OnMouseClick:  Assign=monitoring, Type=Assignment
    hotkey  Id=481037385728, Key=KeyDown=True, KeyName=0, VisuElemId=38
    hotkey  Id=481038434304, Key=KeyName=0, VisuElemId=38
END_VISUALIZATION

// CODESYS_Control_for_Raspberry_Pi/Application/visualization/ups_a2/ups_a2
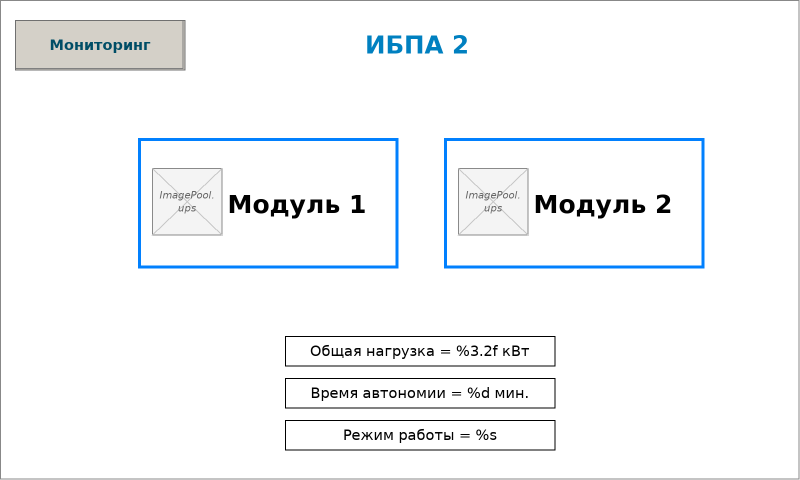
VISUALIZATION ups_a2  // 800x480, background image ImagePool.bg_800
    Rectangle (214,30 406x30), "ИБПА 2"
    Button (15,20 170x50), "Мониторинг"
        OnMouseClick:  Assign=monitoring, Type=Assignment
    Group (138,138 260x115)
        OnMouseClick:  Assign=ups_a2_m1_state, Type=Assignment
        RoundedRectangle (0,0 260x130), colour toggle: InterviewState.MPX_S1_1_State
        Image (14,30 70x67), image: ImagePool.ups
        RoundedRectangle (80,38 158x56), "Модуль 1"
            OnMouseClick:  Assign=ups_s2_m1_state, Type=Assignment
    Group (444,138 260x115)
        OnMouseClick:  Assign=ups_a2_m2_state, Type=Assignment
        RoundedRectangle (0,0 260x130), colour toggle: InterviewState.MPX_S1_2_State
        Image (14,30 70x67), image: ImagePool.ups
        RoundedRectangle (80,38 158x56), "Модуль 2"
            OnMouseClick:  Assign=ups_s2_m1_state, Type=Assignment
    Rectangle (285,336 270x30), "Общая нагрузка = %3.2f кВт", text variable: PLC_PRG.mpx_a2_all_power
    Rectangle (285,378 270x30), "Время автономии = %d мин.", text variable: PLC_PRG.mpx_a2_1_battery_time
    Rectangle (285,420 270x30), "Режим работы = %s", text variable: PLC_PRG.mpx_a2_state_string
    hotkey  Id=481037385728, Key=KeyDown=True, KeyName=0, VisuElemId=38
    hotkey  Id=481038434304, Key=KeyName=0, VisuElemId=38
END_VISUALIZATION

// CODESYS_Control_for_Raspberry_Pi/Application/visualization/ups_a2/ups_a2_m1_params
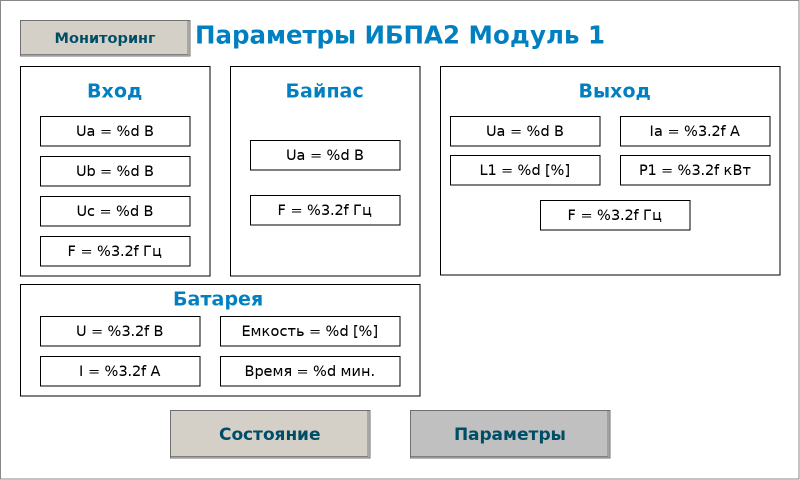
VISUALIZATION ups_a2_m1_params  // 800x480, background image ImagePool.bg_800
    Rectangle (186,20 428x30), "Параметры ИБПА2 Модуль 1"
    Button (170,410 200x48), "Состояние"
        OnMouseClick:  Assign=ups_a2_m1_state, Type=Assignment
    Button (410,410 200x48), "Параметры", pressed state: PLC_PRG.var_true
    Button (20,20 170x36), "Мониторинг"
        OnMouseClick:  Assign=monitoring, Type=Assignment
    Rectangle (20,66 190x210)
    Rectangle (440,66 340x209)
    Rectangle (30,76 170x30), "Вход"
    Rectangle (40,116 150x30), "Ua = %d В", text variable: PLC_PRG.mpx_a2_1_in_v_1
    Rectangle (40,156 150x30), "Ub = %d В", text variable: PLC_PRG.mpx_a2_1_in_v_2
    Rectangle (40,196 150x30), "Uc = %d В", text variable: PLC_PRG.mpx_a2_1_in_v_3
    Rectangle (40,236 150x30), "F = %3.2f Гц", text variable: PLC_PRG.mpx_a2_1_in_freq_real
    Rectangle (230,66 190x210)
    Rectangle (240,76 170x30), "Байпас"
    Rectangle (250,140 150x30), "Ua = %d В", text variable: PLC_PRG.mpx_a2_1_bypass_v_1
    Rectangle (250,195 150x30), "F = %3.2f Гц", text variable: PLC_PRG.mpx_a2_1_bypass_freq_real
    Rectangle (460,76 310x30), "Выход"
    Rectangle (450,116 150x30), "Ua = %d В", text variable: PLC_PRG.mpx_a2_1_output_v_1
    Rectangle (620,116 150x30), "Ia = %3.2f A", text variable: PLC_PRG.mpx_a2_1_output_i_1_real
    Rectangle (450,155 150x30), "L1 = %d [%]", text variable: PLC_PRG.mpx_a2_1_load_ph_1
    Rectangle (620,155 150x30), "P1 = %3.2f кВт", text variable: PLC_PRG.mpx_a2_1_output_active_power_1_real
    Rectangle (540,200 150x30), "F = %3.2f Гц", text variable: PLC_PRG.mpx_a2_1_output_freq_real
    Rectangle (20,284 400x112)
    Rectangle (30,290 376x18), "Батарея"
    Rectangle (40,316 160x30), "U = %3.2f В", text variable: PLC_PRG.mpx_a2_1_battery_voltage_real
    Rectangle (40,356 160x30), "I = %3.2f A", text variable: PLC_PRG.mpx_a2_1_battery_current_real
    Rectangle (220,316 180x30), "Емкость = %d [%]", text variable: PLC_PRG.mpx_a2_1_battery_capacity
    Rectangle (220,356 180x30), "Время = %d мин.", text variable: PLC_PRG.mpx_a2_1_battery_time
    hotkey  Id=481037385728, Key=KeyDown=True, KeyName=0, VisuElemId=7
    hotkey  Id=481038434304, Key=KeyName=0, VisuElemId=7
END_VISUALIZATION

// CODESYS_Control_for_Raspberry_Pi/Application/visualization/ups_a2/ups_a2_m1_state
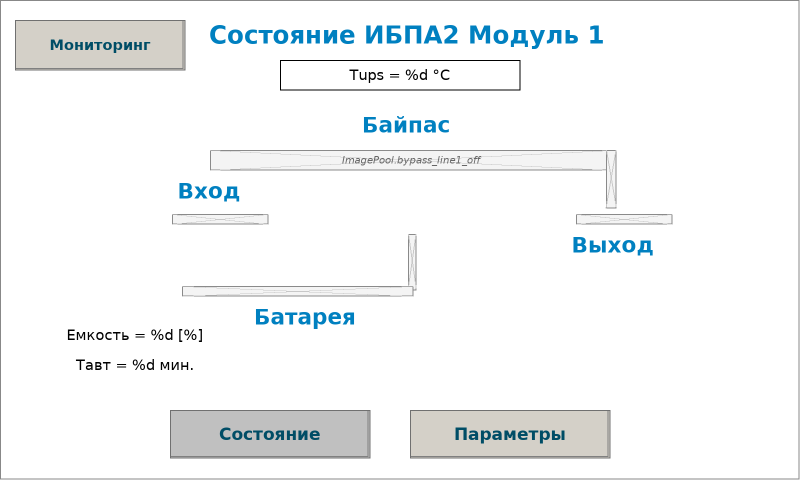
VISUALIZATION ups_a2_m1_state  // 800x480, background image ImagePool.mpx_state_bg
    Rectangle (204,20 406x30), "Состояние ИБПА2 Модуль 1"
    Button (410,410 200x48), "Параметры"
        OnMouseClick:  Assign=ups_a2_m1_params, Type=Assignment
    Button (170,410 200x48), "Состояние", pressed state: PLC_PRG.var_true
    Rectangle (350,110 112x30), "Байпас"
    Rectangle (246,302 118x30), "Батарея"
    Rectangle (166,176 86x30), "Вход"
    Rectangle (560,230 106x30), "Выход"
    Rectangle (280,60 240x30), "Tups = %d °С", text variable: PLC_PRG.mpx_a2_1_temp
    Rectangle (30,320 210x30), "Емкость = %d [%]", text variable: PLC_PRG.mpx_a2_1_battery_capacity
    Rectangle (30,350 210x30), "Tавт = %d мин.", text variable: PLC_PRG.mpx_a2_1_battery_time
    Image (210,150 402x20), image: ImagePool.bypass_line1_off
        p84334746: PLC_PRG.mpx_a2_1_bypass_line_state
    Image (606,150 10x58), image: ImagePool.bypass_arrow_off
        p84334746: PLC_PRG.mpx_a2_1_bypass_arrow_state
    Image (576,214 96x10), image: ImagePool.arrow_off
        p84334746: PLC_PRG.mpx_a2_1_output_state
    Image (172,214 96x10), image: ImagePool.arrow_off
        p84334746: PLC_PRG.mpx_a2_1_input_state
    Image (408,234 8x56), image: ImagePool.battery_arrow_off
        p84334746: PLC_PRG.mpx_a2_1_battery_arrow_state
    Image (182,286 231x10), image: ImagePool.battery_line_off
        p84334746: PLC_PRG.mpx_a2_1_battery_line_state
    Button (15,20 170x50), "Мониторинг"
        OnMouseClick:  Assign=monitoring, Type=Assignment
    hotkey  Id=481037385728, Key=KeyDown=True, KeyName=0, VisuElemId=38
    hotkey  Id=481038434304, Key=KeyName=0, VisuElemId=38
END_VISUALIZATION

// CODESYS_Control_for_Raspberry_Pi/Application/visualization/ups_a2/ups_a2_m2_params
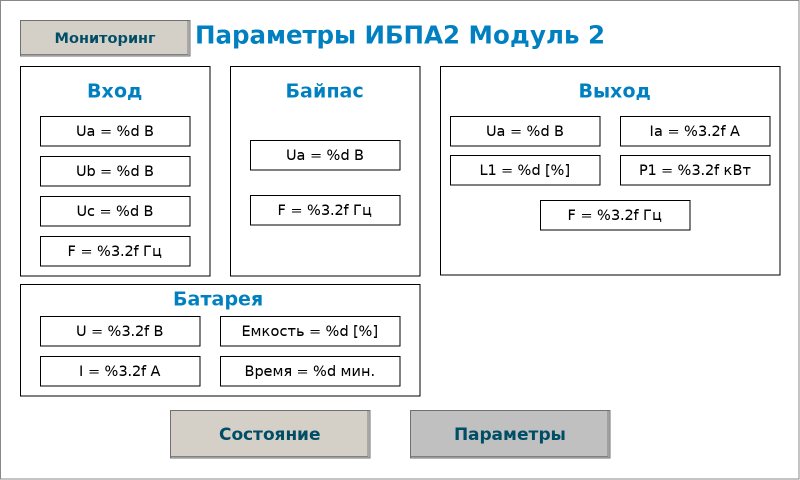
VISUALIZATION ups_a2_m2_params  // 800x480, background image ImagePool.bg_800
    Rectangle (186,20 428x30), "Параметры ИБПА2 Модуль 2"
    Button (170,410 200x48), "Состояние"
        OnMouseClick:  Assign=ups_a2_m2_state, Type=Assignment
    Button (410,410 200x48), "Параметры", pressed state: PLC_PRG.var_true
    Button (20,20 170x36), "Мониторинг"
        OnMouseClick:  Assign=monitoring, Type=Assignment
    Rectangle (20,66 190x210)
    Rectangle (440,66 340x209)
    Rectangle (30,76 170x30), "Вход"
    Rectangle (40,116 150x30), "Ua = %d В", text variable: PLC_PRG.mpx_a2_2_in_v_1
    Rectangle (40,156 150x30), "Ub = %d В", text variable: PLC_PRG.mpx_a2_2_in_v_2
    Rectangle (40,196 150x30), "Uc = %d В", text variable: PLC_PRG.mpx_a2_2_in_v_3
    Rectangle (40,236 150x30), "F = %3.2f Гц", text variable: PLC_PRG.mpx_a2_2_in_freq_real
    Rectangle (230,66 190x210)
    Rectangle (240,76 170x30), "Байпас"
    Rectangle (250,140 150x30), "Ua = %d В", text variable: PLC_PRG.mpx_a2_2_bypass_v_1
    Rectangle (250,195 150x30), "F = %3.2f Гц", text variable: PLC_PRG.mpx_a2_2_bypass_freq_real
    Rectangle (460,76 310x30), "Выход"
    Rectangle (450,116 150x30), "Ua = %d В", text variable: PLC_PRG.mpx_a2_2_output_v_1
    Rectangle (620,116 150x30), "Ia = %3.2f A", text variable: PLC_PRG.mpx_a2_2_output_i_1_real
    Rectangle (450,155 150x30), "L1 = %d [%]", text variable: PLC_PRG.mpx_a2_2_load_ph_1
    Rectangle (620,155 150x30), "P1 = %3.2f кВт", text variable: PLC_PRG.mpx_a2_2_output_active_power_1_real
    Rectangle (540,200 150x30), "F = %3.2f Гц", text variable: PLC_PRG.mpx_a2_2_output_freq_real
    Rectangle (20,284 400x112)
    Rectangle (30,290 376x18), "Батарея"
    Rectangle (40,316 160x30), "U = %3.2f В", text variable: PLC_PRG.mpx_a2_2_battery_voltage_real
    Rectangle (40,356 160x30), "I = %3.2f A", text variable: PLC_PRG.mpx_a2_2_battery_current_real
    Rectangle (220,316 180x30), "Емкость = %d [%]", text variable: PLC_PRG.mpx_a2_2_battery_capacity
    Rectangle (220,356 180x30), "Время = %d мин.", text variable: PLC_PRG.mpx_a2_2_battery_time
    hotkey  Id=481037385728, Key=KeyDown=True, KeyName=0, VisuElemId=7
    hotkey  Id=481038434304, Key=KeyName=0, VisuElemId=7
END_VISUALIZATION

// CODESYS_Control_for_Raspberry_Pi/Application/visualization/ups_a2/ups_a2_m2_state
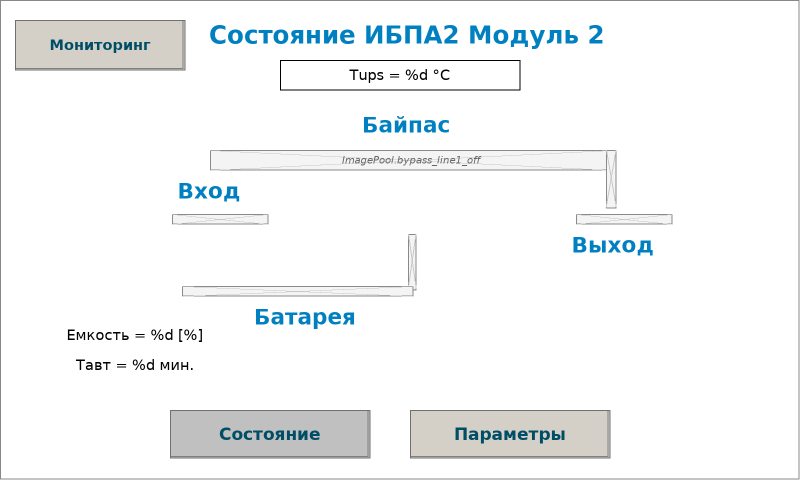
VISUALIZATION ups_a2_m2_state  // 800x480, background image ImagePool.mpx_state_bg
    Rectangle (204,20 406x30), "Состояние ИБПА2 Модуль 2"
    Button (410,410 200x48), "Параметры"
        OnMouseClick:  Assign=ups_a2_m2_params, Type=Assignment
    Button (170,410 200x48), "Состояние", pressed state: PLC_PRG.var_true
    Rectangle (350,110 112x30), "Байпас"
    Rectangle (246,302 118x30), "Батарея"
    Rectangle (166,176 86x30), "Вход"
    Rectangle (560,230 106x30), "Выход"
    Rectangle (280,60 240x30), "Tups = %d °С", text variable: PLC_PRG.mpx_a2_2_temp
    Rectangle (30,320 210x30), "Емкость = %d [%]", text variable: PLC_PRG.mpx_a2_2_battery_capacity
    Rectangle (30,350 210x30), "Tавт = %d мин.", text variable: PLC_PRG.mpx_a2_2_battery_time
    Image (210,150 402x20), image: ImagePool.bypass_line1_off
        p84334746: PLC_PRG.mpx_a2_2_bypass_line_state
    Image (606,150 10x58), image: ImagePool.bypass_arrow_off
        p84334746: PLC_PRG.mpx_a2_2_bypass_arrow_state
    Image (576,214 96x10), image: ImagePool.arrow_off
        p84334746: PLC_PRG.mpx_a2_2_output_state
    Image (172,214 96x10), image: ImagePool.arrow_off
        p84334746: PLC_PRG.mpx_a2_2_input_state
    Image (408,234 8x56), image: ImagePool.battery_arrow_off
        p84334746: PLC_PRG.mpx_a2_2_battery_arrow_state
    Image (182,286 231x10), image: ImagePool.battery_line_off
        p84334746: PLC_PRG.mpx_a2_2_battery_line_state
    Button (15,20 170x50), "Мониторинг"
        OnMouseClick:  Assign=monitoring, Type=Assignment
    hotkey  Id=481037385728, Key=KeyDown=True, KeyName=0, VisuElemId=38
    hotkey  Id=481038434304, Key=KeyName=0, VisuElemId=38
END_VISUALIZATION

// CODESYS_Control_for_Raspberry_Pi/Application/visualization/climate_log
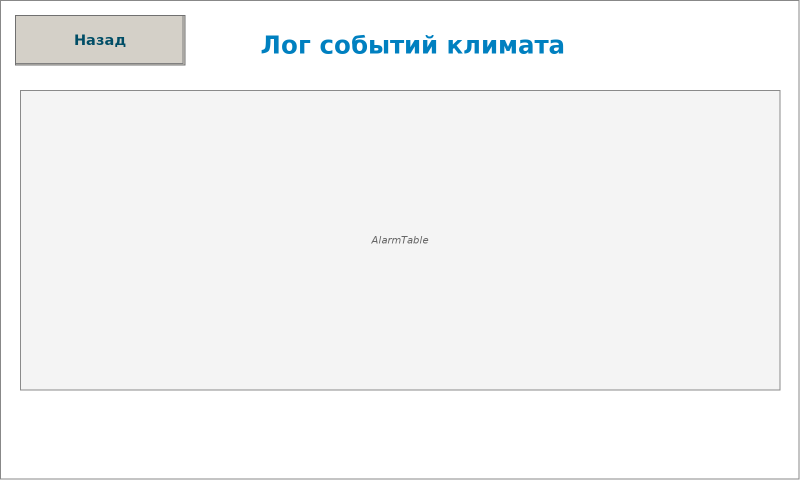
VISUALIZATION climate_log  // 800x480, background image ImagePool.bg_800
    Button (15,15 170x50), "Назад"
        OnMouseClick:  Assign=climate, Type=Previous
    Rectangle (210,30 406x30), "Лог событий климата"
    AlarmTable (20,90 760x300)
        Column[0]: ColumnTitle=Временная отметка
        Column[1]: ColumnTitle=Сообщение
        p1521930926: ClimateGroup
        p1663851261: __All
        p3266827225: PLC_PRG.var_true
    hotkey  Id=481037385728, Key=KeyDown=True, KeyName=0, VisuElemId=1
    hotkey  Id=481038434304, Key=KeyName=0, VisuElemId=1
END_VISUALIZATION

// CODESYS_Control_for_Raspberry_Pi/Application/visualization/more
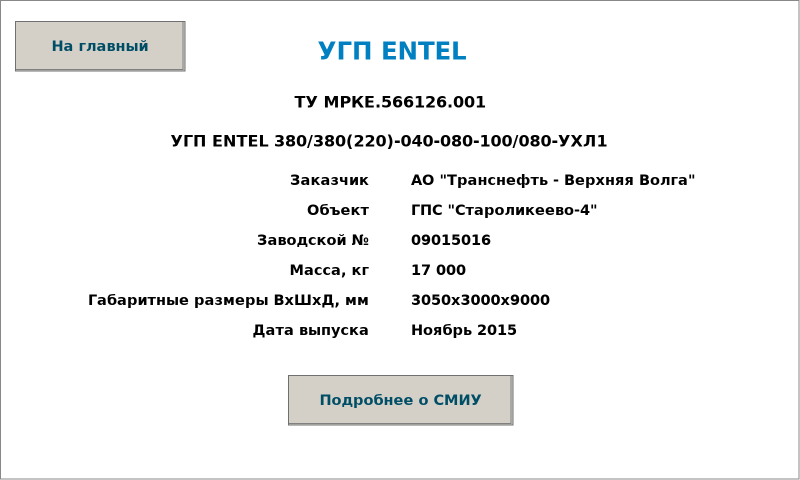
VISUALIZATION more  // 800x480, background image ImagePool.bg_800
    Rectangle (189,36 406x30), "УГП ENTEL"
    Button (15,21 170x50), "На главный"
        OnMouseClick:  Assign=main, Type=Assignment
    Button (288,375 225x50), "Подробнее о СМИУ"
        OnMouseClick:  Assign=info, Type=Assignment
    Label (213,87 355x30), "ТУ МРКЕ.566126.001"
    Label (186,126 406x30), "УГП ENTEL 380/380(220)-040-080-100/080-УХЛ1"
    Label (276,165 96x30), "Заказчик"
    Label (276,195 96x30), "Объект"
    Label (246,225 126x30), "Заводской №"
    Label (276,255 96x30), "Масса, кг"
    Label (96,285 276x30), "Габаритные размеры ВхШхД, мм"
    Label (201,315 171x30), "Дата выпуска"
    Label (408,165 309x30), "АО "Транснефть - Верхняя Волга""
    Label (408,195 228x30), "ГПС "Староликеево-4""
    Label (408,225 114x30), "09015016"
    Label (408,255 120x30), "17 000"
    Label (408,285 165x30), "3050х3000х9000"
    Label (408,315 126x30), "Ноябрь 2015"
    hotkey  Id=481037385728, Key=KeyDown=True, KeyName=0, VisuElemId=3
    hotkey  Id=481038434304, Key=KeyName=0, VisuElemId=3
    hotkey  Id=481037385728, Key=KeyDown=True, KeyName=0, VisuElemId=5
    hotkey  Id=481038434304, Key=KeyName=0, VisuElemId=5
END_VISUALIZATION

(* text list AlarmGroup (id | default)
  95 | Отсутствует напряжение на выходе ИБПА 2
  94 | Отсутствует напряжение на выходе ИБПА 1
  93 | Отсутствует напряжение на выходе ИБПС 2
  92 | Отсутствует напряжение на выходе ИБПС 1
  91 | Отсутствует напряжение на входе ИБПА 2
  90 | Отсутствует напряжение на входе ИБПА 1
  89 | Отсутствует напряжение на входе ИБПС 2
  88 | Отсутствует напряжение на входе ИБПС 1
  87 | Отключен выходной автомат ИБПС 2
  86 | Отсутствует напряжения на выходе ИБПС 2 модуль 4 (1ф.)
  85 | Отключен выходной автомат ИБПС 1
  84 | Отсутствует напряжения на выходе ИБПС 2 модуль 4 (3ф.)
  83 | Отсутствует напряжения на выходе ИБПС 2 модуль 4 (2ф.)
  82 | Отсутствует напряжения на выходе ИБПС 2 модуль 4 (1ф.)
  81 | Отсутствует напряжения на выходе ИБПС 2 модуль 3 (3ф.)
  80 | Отсутствует напряжения на выходе ИБПС 2 модуль 3 (2ф.)
  79 | Отсутствует напряжения на выходе ИБПС 2 модуль 3 (1ф.)
  78 | Отсутствует напряжения на выходе ИБПС 2 модуль 2 (3ф.)
  77 | Отсутствует напряжения на выходе ИБПС 2 модуль 2 (2ф.)
  76 | Отсутствует напряжения на выходе ИБПС 2 модуль 2 (1ф.)
  75 | Отсутствует напряжения на выходе ИБПС 2 модуль 1 (3ф.)
  74 | Отсутствует напряжения на выходе ИБПС 2 модуль 1 (2ф.)
  73 | Отсутствует напряжения на выходе ИБПС 2 модуль 1 (1ф.)
  72 | Отсутствует напряжения на выходе ИБПС 1 модуль 4 (3ф.)
  71 | Отсутствует напряжения на выходе ИБПС 1 модуль 4 (2ф.)
  70 | Отсутствует напряжения на выходе ИБПС 1 модуль 4 (1ф.)
  69 | Отсутствует напряжения на выходе ИБПС 1 модуль 3 (3ф.)
  68 | Отсутствует напряжения на выходе ИБПС 1 модуль 3 (2ф.)
  67 | Отсутствует напряжения на выходе ИБПС 1 модуль 3 (1ф.)
  66 | Отсутствует напряжения на выходе ИБПС 1 модуль 2 (3ф.)
  65 | Отсутствует напряжения на выходе ИБПС 1 модуль 2 (2ф.)
  64 | Отсутствует напряжения на выходе ИБПС 1 модуль 2 (1ф.)
  63 | Отсутствует напряжения на выходе ИБПС 1 модуль 1 (3ф.)
  62 | Отсутствует напряжения на выходе ИБПС 1 модуль 1 (2ф.)
  61 | Отсутствует напряжения на выходе ИБПС 1 модуль 1 (1ф.)
  60 | Отсутствует напряжения на выходе ИБПА 2 модуль 2
  59 | Отсутствует напряжения на выходе ИБПА 2 модуль 1
  58 | Отсутствует напряжения на выходе ИБПА 1 модуль 2
  57 | Отсутствует напряжения на выходе ИБПА 1 модуль 1
  56 | Авария ИБПС 2 модуль 4
  55 | Авария ИБПС 2 модуль 3
  54 | Авария ИБПС 2 модуль 2
  53 | Авария ИБПС 2 модуль 1
  52 | Авария ИБПС 1 модуль 4
  51 | Авария ИБПС 1 модуль 3
  50 | Авария ИБПС 1 модуль 2
  49 | Авария ИБПС 1 модуль 1
  48 | Авария ИБПА 2 модуль 2
  47 | Авария ИБПА 2 модуль 1
  46 | Авария ИБПА 1 модуль 2
  45 | Авария ИБПА 1 модуль 1
  44 | Отсутствует напряжение на входе ИБПC 2 модуль 4 (3 ф.)
  43 | Отсутствует напряжение на входе ИБПC 2 модуль 4 (2 ф.)
  42 | Отсутствует напряжение на входе ИБПC 2 модуль 4 (1 ф.)
  41 | Отсутствует напряжение на входе ИБПC 2 модуль 3 (3 ф.)
  40 | Отсутствует напряжение на входе ИБПC 2 модуль 3 (2 ф.)
  39 | Отсутствует напряжение на входе ИБПC 2 модуль 3 (1 ф.)
  38 | Отсутствует напряжение на входе ИБПC 2 модуль 2 (3 ф.)
  37 | Отсутствует напряжение на входе ИБПC 2 модуль 2 (2 ф.)
  36 | Отсутствует напряжение на входе ИБПC 2 модуль 2 (1 ф.)
  35 | Отсутствует напряжение на входе ИБПC 2 модуль 1 (3 ф.)
  34 | Отсутствует напряжение на входе ИБПC 2 модуль 1 (2 ф.)
  33 | Отсутствует напряжение на входе ИБПC 2 модуль 1 (1 ф.)
  32 | Отсутствует напряжение на входе ИБПC 1 модуль 4 (3 ф.)
  31 | Отсутствует напряжение на входе ИБПC 1 модуль 4 (2 ф.)
  30 | Отсутствует напряжение на входе ИБПC 1 модуль 4 (1 ф.)
  29 | Отсутствует напряжение на входе ИБПC 1 модуль 3 (3 ф.)
  28 | Отсутствует напряжение на входе ИБПC 1 модуль 3 (2 ф.)
  27 | Отсутствует напряжение на входе ИБПC 1 модуль 3 (1 ф.)
  26 | Отсутствует напряжение на входе ИБПC 1 модуль 2 (3 ф.)
  25 | Отсутствует напряжение на входе ИБПC 1 модуль 2 (2 ф.)
  24 | Отсутствует напряжение на входе ИБПC 1 модуль 1 (3 ф.)
  23 | Отсутствует напряжение на входе ИБПC 1 модуль 2 (1 ф.)
  22 | Отсутствует напряжение на входе ИБПC 1 модуль 1 (2 ф.)
  21 | Отсутствует напряжение на входе ИБПC 1 модуль 1 (1 ф.)
  20 | Отсутствует напряжение на входе ИБПА 2 модуль 2 (3 ф.)
  19 | Отсутствует напряжение на входе ИБПА 2 модуль 2 (2 ф.)
  18 | Отсутствует напряжение на входе ИБПА 2 модуль 2 (1 ф.)
  17 | Отсутствует напряжение на входе ИБПА 2 модуль 1 (3 ф.)
  16 | Отсутствует напряжение на входе ИБПА 2 модуль 1 (2 ф.)
  15 | Отсутствует напряжение на входе ИБПА 2 модуль 1 (1 ф.)
  14 | Отсутствует напряжение на входе ИБПА 1 модуль 2 (3 ф.)
  13 | Отсутствует напряжение на входе ИБПА 1 модуль 2 (2 ф.)
  12 | Отсутствует напряжение на входе ИБПА 1 модуль 2 (1 ф.)
  11 | Отсутствует напряжение на входе ИБПА 1 модуль 1 (3 ф.)
  10 | Отсутствует напряжение на входе ИБПА 1 модуль 1 (2 ф.)
  9 | 
  8 | Отсутствует напряжение на входе ИБПА 1 модуль 1 (1 ф.)
  7 | Отсутствует напряжение на шине ГП ШАСН
  6 | Отсутствует напряжение на шине БП ШАСН
  5 | Отсутствует напряжение на ГП 2 ЩРПС
  4 | Отсутствует напряжение на ГП 1 ЩРПС
  3 | Отсутствует напряжение на резервном вводе ШАСН
  2 | Отсутствует напряжение на основном вводе ШАСН
  1 | Отсутствует напряжение на резервном вводе ЩРПА
  0 | Отсутствует напряжение на основном вводе ЩРПА
   |  *)

(* text list ClimateGroup (id | default)
  11 | Обогрев дверей выключен
  10 | Обогрев дверей включен
  9 | Кондиционеры выключены
  8 | Кондиционеры включены
  7 | Вентиляторы выключены
  6 | Вентиляторы включены
  5 | Заслонка закрыта
  4 | Заслонка открыта
  3 | Автоматика выключена
  2 | Обогрев выключен
  1 | Автоматика включена
  0 | Обогрев включен
   |  *)
